FUNCTION F_WORDFromBytes : WORD
VAR_INPUT
    B1 : BYTE;
    B0 : BYTE;
END_VAR

F_WORDFromBytes := SHL(BYTE_TO_WORD(B1),8) OR BYTE_TO_WORD(B0);

END_FUNCTION

(* stored: Version 1.1.0.1, ProductVersion 3.1.4022.18
   POU F_WORDFromBytes: Id {d1564ac0-d69f-409c-b1e8-deaeae45b009}, SpecialFunc None *)
